(* Logix 5000 project; controller Sucrose_Main Emulate 5570 rev 20.12; software revision 20.01; part 25 of 30 *)
(* tags used below, declared in another part *)
   Alarm_ACK_Master_Timer : TIMER;
   CIPRemote : Area_Program;
   CR13582_AOI : QSI_Discrete_Device;   // CR-13582 SUCROSE RECEIVING PUMP #1 SEAL WATER VALVE
   CR13584_AOI : QSI_Discrete_Device;   // CR-13584 SUCROSE RECEIVING PUMP #2 SEAL WATER VALVE
   DI_E25_2 : ALIAS FOR FLX_E25:2:I;   // Discrete Input EN2T_FLX 192.168.1.25
   DI_E25_3 : ALIAS FOR FLX_E25:3:I;   // Discrete Input EN2T_FLX 192.168.1.25
   DO_E25_4 : ALIAS FOR FLX_E25:4:O;   // Discrete Output EN2T_FLX 192.168.1.25
   DO_E25_5 : ALIAS FOR FLX_E25:5:O;   // Discrete Output EN2T_FLX 192.168.1.25
   FV230001_AOI : QSI_Flow_Valve;   // FV-23-00-01 LAUNCH PIG VALVE V1
   FV230002_AOI : QSI_Flow_Valve;   // FV-23-00-02 LAUNCH PIG VALVE V2
   FV2300031_AOI : QSI_Flow_Valve;   // FV-23-00-03_1 MOVE PIG BACKWARDS INTO CIP/PRODUCTION POSITION
   FV2300032_AOI : QSI_Flow_Valve;   // FV-23-00-03_2 MOVE PIG FORWARD INTO LAUNCHING POSITION
   FV230004_AOI : QSI_Flow_Valve;   // FV-23-00-04 PIG RETENTION CYLINDER V4.1
   FV230005_AOI : QSI_Flow_Valve;   // FV-23-00-05 PIG RETENTION CYLINDER V4.2
   FV230010_AOI : QSI_Flow_Valve;   // FV-23-00-10-O RECEIVING PUMP #1 TO SUCROSE VALVE MANIFOLD MIX PROOF VALVE OPEN
   FV230020_AOI : QSI_Flow_Valve;   // FV-23-00-20-O RECEIVING PUMP #2 TO SUCROSE VALVE MANIFOLD MIX PROOF VALVE OPEN
   IO_Check : BOOL;
   P230010_AOI : PF525_VFD_E_ENET;   // P-23-00-10 RECEIVING PUMP 1
   P230020_AOI : PF525_VFD_E_ENET;   // P-23-00-20 RECEIVING PUMP 2
   PBL1604002_AOI : QSI_Discrete_Device;   // PBL-16040-02 E-STOP CIRCUIT RESET LIGHT
   PSV230010_AOI : QSI_Flow_Valve;
   PSV230020_AOI : QSI_Flow_Valve;
   Sucrose_MM_Enable : BOOL;
   SucroseCIP_RECEIVING2_REMOTE : CIP_REMOTE;
   SucroseCIP_RECEIVING_LINE_REMOTE : CIP_REMOTE;
   SucroseCIP_RECEIVING_REMOTE : CIP_REMOTE;
   SucroseReceiving : Area_Program;
   TMR_SLOW_PLS1 : TIMER;
   TMR_SLOW_PLS2 : TIMER;

PROGRAM ReceivingArea_EN2T_IO_Discrete_DO_E25_4   (* main routine MainRoutine *)

ROUTINE _00_FV230001   (* ladder *)
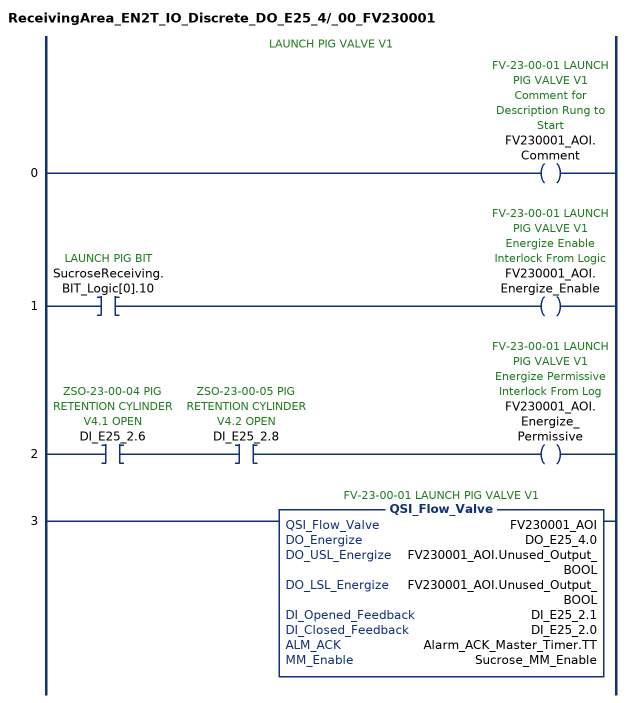
   // LAUNCH PIG VALVE V1
   0: OTE(FV230001_AOI.Comment);
   1: XIC(SucroseReceiving.BIT_Logic[0].10)OTE(FV230001_AOI.Energize_Enable);
   2: XIC(DI_E25_2.6)XIC(DI_E25_2.8)OTE(FV230001_AOI.Energize_Permissive);
   3: QSI_Flow_Valve(FV230001_AOI,DO_E25_4.0,FV230001_AOI.Unused_Output_BOOL,FV230001_AOI.Unused_Output_BOOL,DI_E25_2.1,DI_E25_2.0,Alarm_ACK_Master_Timer.TT,Sucrose_MM_Enable);
END_ROUTINE

ROUTINE _01_FV230002   (* ladder *)
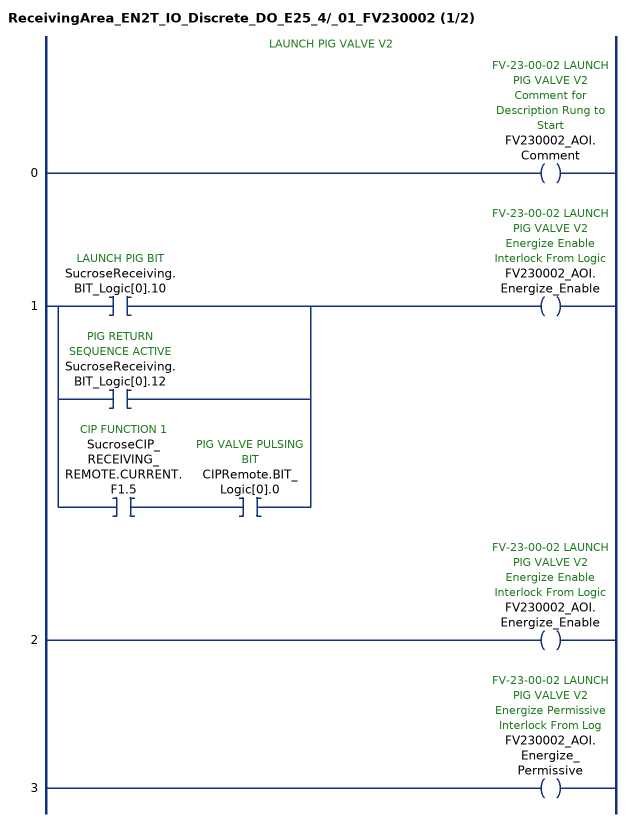
   // LAUNCH PIG VALVE V2
   0: OTE(FV230002_AOI.Comment);
   1: [XIC(SucroseReceiving.BIT_Logic[0].10) ,XIC(SucroseReceiving.BIT_Logic[0].12) ,XIC(SucroseCIP_RECEIVING_REMOTE.CURRENT.F1.5) XIC(CIPRemote.BIT_Logic[0].0) ]OTE(FV230002_AOI.Energize_Enable);
   2: OTE(FV230002_AOI.Energize_Enable);
   3: OTE(FV230002_AOI.Energize_Permissive);
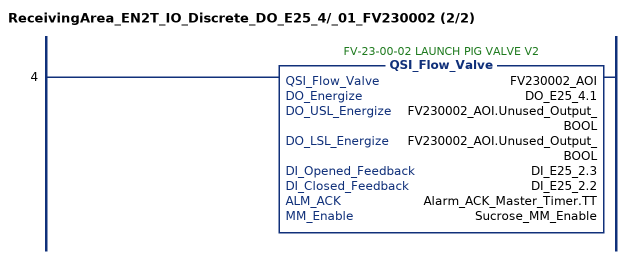
   4: QSI_Flow_Valve(FV230002_AOI,DO_E25_4.1,FV230002_AOI.Unused_Output_BOOL,FV230002_AOI.Unused_Output_BOOL,DI_E25_2.3,DI_E25_2.2,Alarm_ACK_Master_Timer.TT,Sucrose_MM_Enable);
END_ROUTINE

ROUTINE _02_FV230004   (* ladder *)
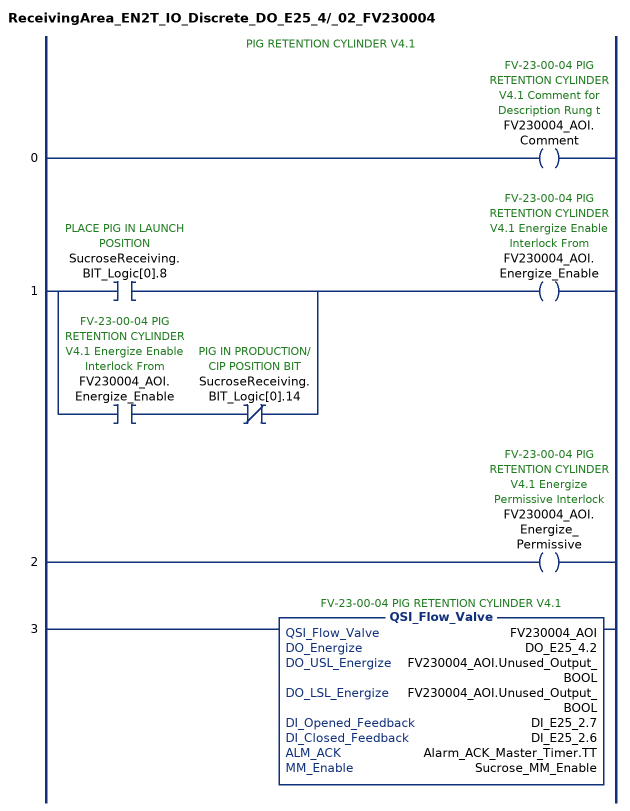
   // PIG RETENTION CYLINDER V4.1
   0: OTE(FV230004_AOI.Comment);
   1: [XIC(SucroseReceiving.BIT_Logic[0].8) ,XIC(FV230004_AOI.Energize_Enable) XIO(SucroseReceiving.BIT_Logic[0].14) ]OTE(FV230004_AOI.Energize_Enable);
   2: OTE(FV230004_AOI.Energize_Permissive);
   3: QSI_Flow_Valve(FV230004_AOI,DO_E25_4.2,FV230004_AOI.Unused_Output_BOOL,FV230004_AOI.Unused_Output_BOOL,DI_E25_2.7,DI_E25_2.6,Alarm_ACK_Master_Timer.TT,Sucrose_MM_Enable);
END_ROUTINE

ROUTINE _03_FV2300031   (* ladder *)
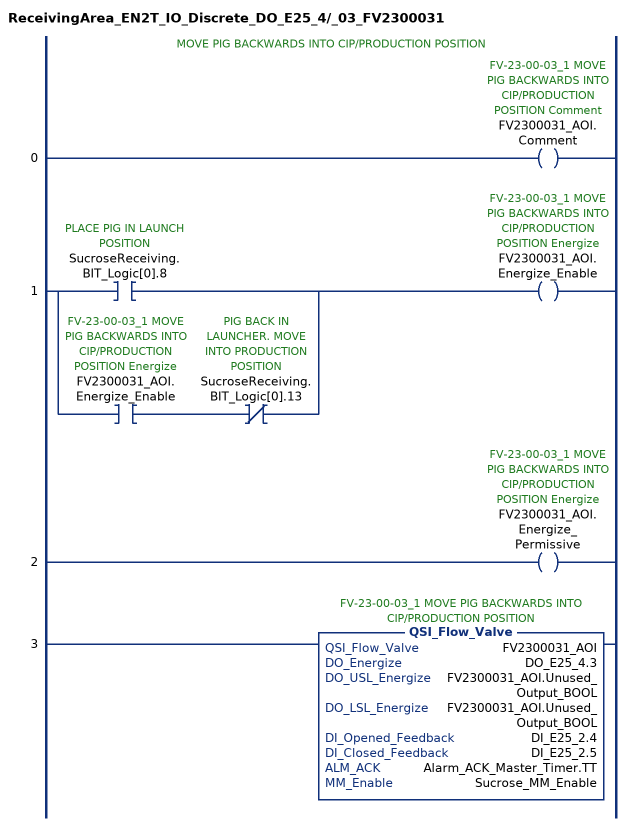
   // MOVE PIG BACKWARDS INTO CIP/PRODUCTION POSITION
   0: OTE(FV2300031_AOI.Comment);
   1: [XIC(SucroseReceiving.BIT_Logic[0].8) ,XIC(FV2300031_AOI.Energize_Enable) XIO(SucroseReceiving.BIT_Logic[0].13) ]OTE(FV2300031_AOI.Energize_Enable);
   2: OTE(FV2300031_AOI.Energize_Permissive);
   3: QSI_Flow_Valve(FV2300031_AOI,DO_E25_4.3,FV2300031_AOI.Unused_Output_BOOL,FV2300031_AOI.Unused_Output_BOOL,DI_E25_2.4,DI_E25_2.5,Alarm_ACK_Master_Timer.TT,Sucrose_MM_Enable);
END_ROUTINE

ROUTINE _04_FV230005   (* ladder *)
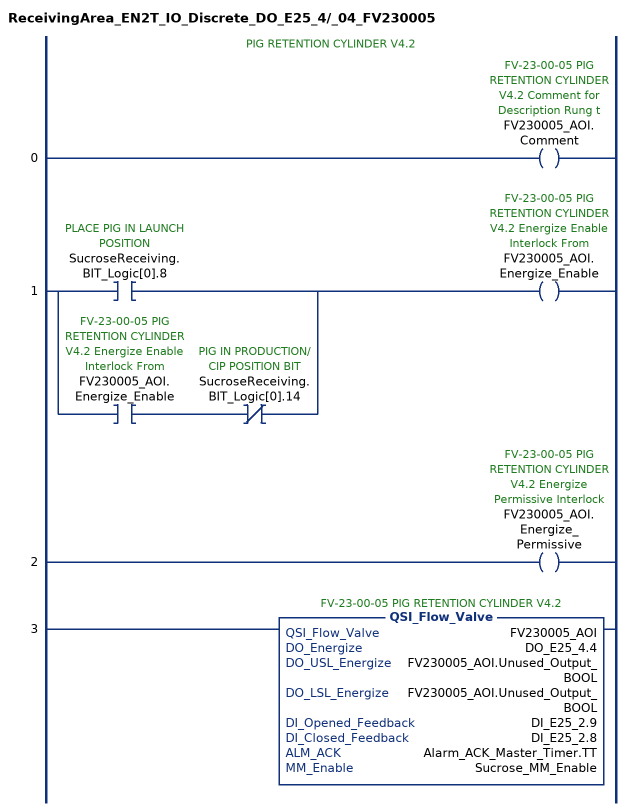
   // PIG RETENTION CYLINDER V4.2
   0: OTE(FV230005_AOI.Comment);
   1: [XIC(SucroseReceiving.BIT_Logic[0].8) ,XIC(FV230005_AOI.Energize_Enable) XIO(SucroseReceiving.BIT_Logic[0].14) ]OTE(FV230005_AOI.Energize_Enable);
   2: OTE(FV230005_AOI.Energize_Permissive);
   3: QSI_Flow_Valve(FV230005_AOI,DO_E25_4.4,FV230005_AOI.Unused_Output_BOOL,FV230005_AOI.Unused_Output_BOOL,DI_E25_2.9,DI_E25_2.8,Alarm_ACK_Master_Timer.TT,Sucrose_MM_Enable);
END_ROUTINE

ROUTINE _05_FV2300032   (* ladder *)
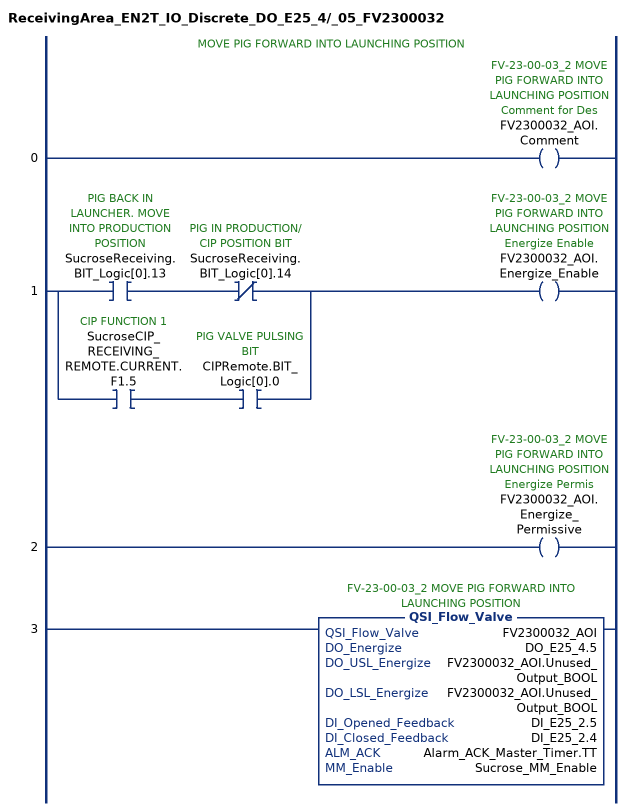
   // MOVE PIG FORWARD INTO LAUNCHING POSITION
   0: OTE(FV2300032_AOI.Comment);
   1: [XIC(SucroseReceiving.BIT_Logic[0].13) XIO(SucroseReceiving.BIT_Logic[0].14) ,XIC(SucroseCIP_RECEIVING_REMOTE.CURRENT.F1.5) XIC(CIPRemote.BIT_Logic[0].0) ]OTE(FV2300032_AOI.Energize_Enable);
   2: OTE(FV2300032_AOI.Energize_Permissive);
   3: QSI_Flow_Valve(FV2300032_AOI,DO_E25_4.5,FV2300032_AOI.Unused_Output_BOOL,FV2300032_AOI.Unused_Output_BOOL,DI_E25_2.5,DI_E25_2.4,Alarm_ACK_Master_Timer.TT,Sucrose_MM_Enable);
END_ROUTINE

ROUTINE _10_PSV230010   (* ladder *)
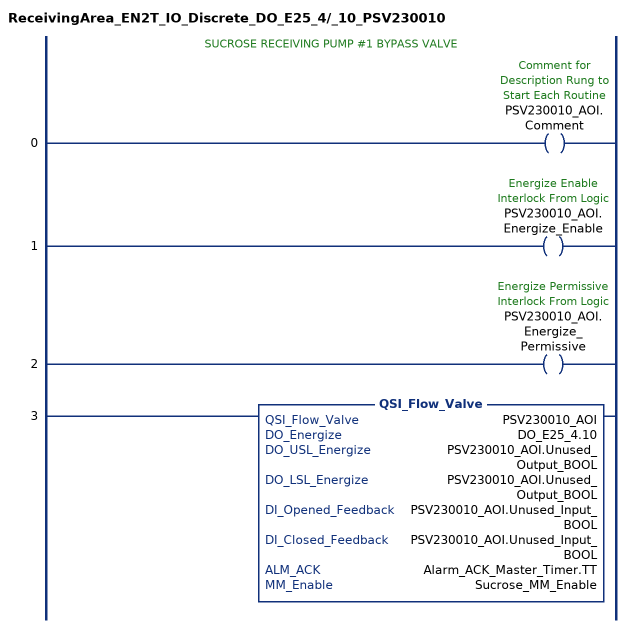
   // SUCROSE RECEIVING PUMP #1 BYPASS VALVE
   0: OTE(PSV230010_AOI.Comment);
   1: OTE(PSV230010_AOI.Energize_Enable);
   2: OTE(PSV230010_AOI.Energize_Permissive);
   3: QSI_Flow_Valve(PSV230010_AOI,DO_E25_4.10,PSV230010_AOI.Unused_Output_BOOL,PSV230010_AOI.Unused_Output_BOOL,PSV230010_AOI.Unused_Input_BOOL,PSV230010_AOI.Unused_Input_BOOL,Alarm_ACK_Master_Timer.TT,Sucrose_MM_Enable);
END_ROUTINE

ROUTINE _11_PSV230020   (* ladder *)
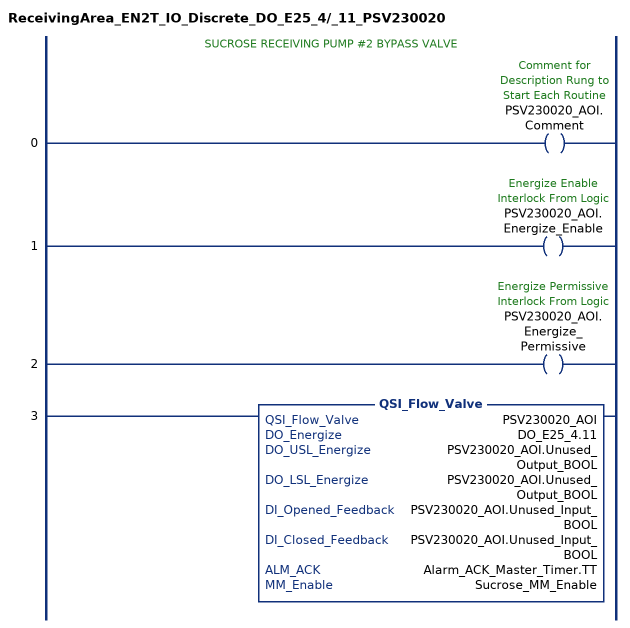
   // SUCROSE RECEIVING PUMP #2 BYPASS VALVE
   0: OTE(PSV230020_AOI.Comment);
   1: OTE(PSV230020_AOI.Energize_Enable);
   2: OTE(PSV230020_AOI.Energize_Permissive);
   3: QSI_Flow_Valve(PSV230020_AOI,DO_E25_4.11,PSV230020_AOI.Unused_Output_BOOL,PSV230020_AOI.Unused_Output_BOOL,PSV230020_AOI.Unused_Input_BOOL,PSV230020_AOI.Unused_Input_BOOL,Alarm_ACK_Master_Timer.TT,Sucrose_MM_Enable);
END_ROUTINE

ROUTINE MainRoutine   (* ladder *)
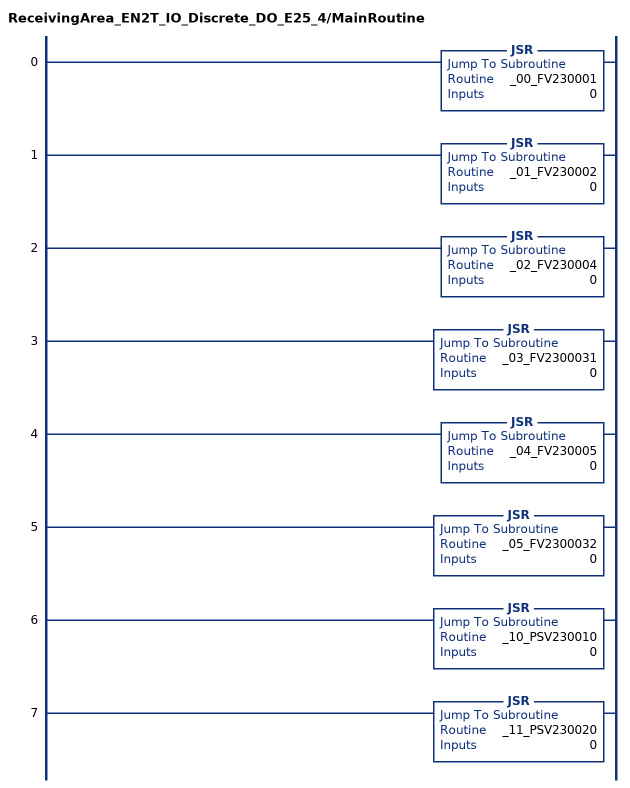
   0: JSR(_00_FV230001,0);
   1: JSR(_01_FV230002,0);
   2: JSR(_02_FV230004,0);
   3: JSR(_03_FV2300031,0);
   4: JSR(_04_FV230005,0);
   5: JSR(_05_FV2300032,0);
   6: JSR(_10_PSV230010,0);
   7: JSR(_11_PSV230020,0);
END_ROUTINE
END_PROGRAM

PROGRAM ReceivingArea_EN2T_IO_Discrete_DO_E25_5   (* main routine MainRoutine *)

ROUTINE _00_FV230010   (* ladder *)
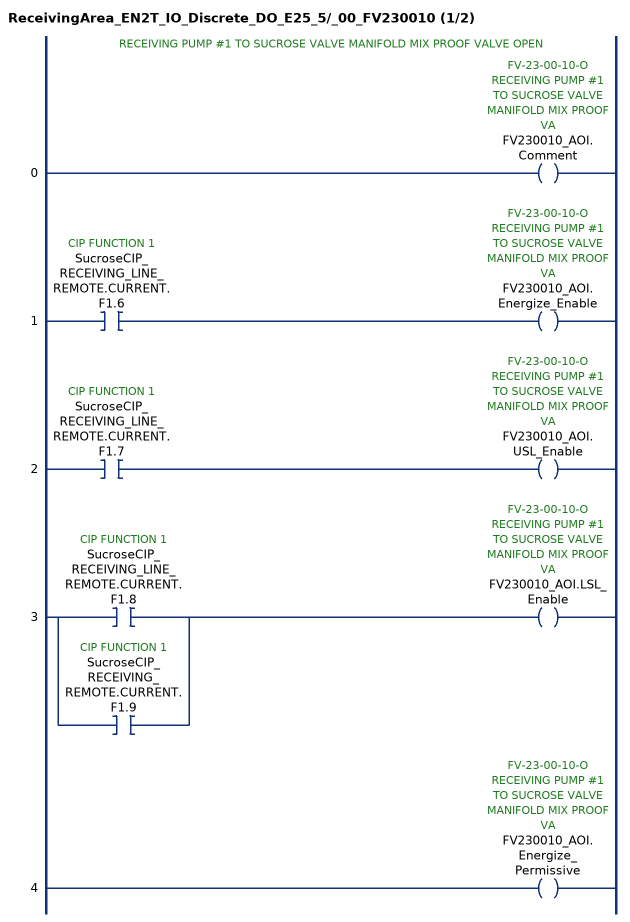
   // RECEIVING PUMP #1 TO SUCROSE VALVE MANIFOLD MIX PROOF VALVE OPEN
   0: OTE(FV230010_AOI.Comment);
   1: XIC(SucroseCIP_RECEIVING_LINE_REMOTE.CURRENT.F1.6)OTE(FV230010_AOI.Energize_Enable);
   2: XIC(SucroseCIP_RECEIVING_LINE_REMOTE.CURRENT.F1.7)OTE(FV230010_AOI.USL_Enable);
   3: [XIC(SucroseCIP_RECEIVING_LINE_REMOTE.CURRENT.F1.8) ,XIC(SucroseCIP_RECEIVING_REMOTE.CURRENT.F1.9) ]OTE(FV230010_AOI.LSL_Enable);
   4: OTE(FV230010_AOI.Energize_Permissive);
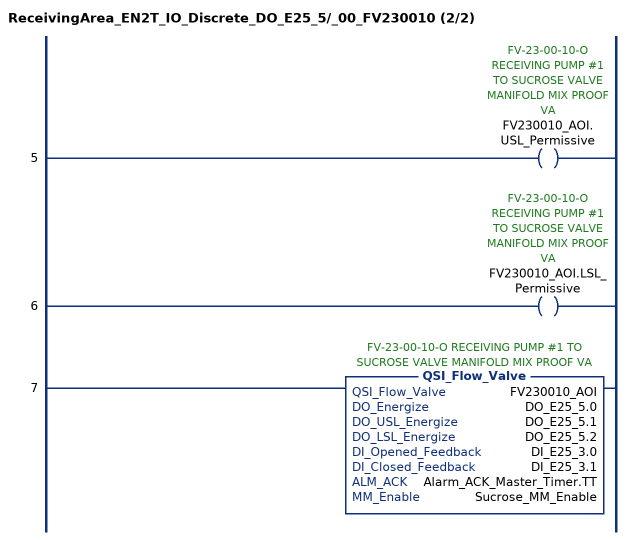
   5: OTE(FV230010_AOI.USL_Permissive);
   6: OTE(FV230010_AOI.LSL_Permissive);
   7: QSI_Flow_Valve(FV230010_AOI,DO_E25_5.0,DO_E25_5.1,DO_E25_5.2,DI_E25_3.0,DI_E25_3.1,Alarm_ACK_Master_Timer.TT,Sucrose_MM_Enable);
END_ROUTINE

ROUTINE _03_FV230020   (* ladder *)
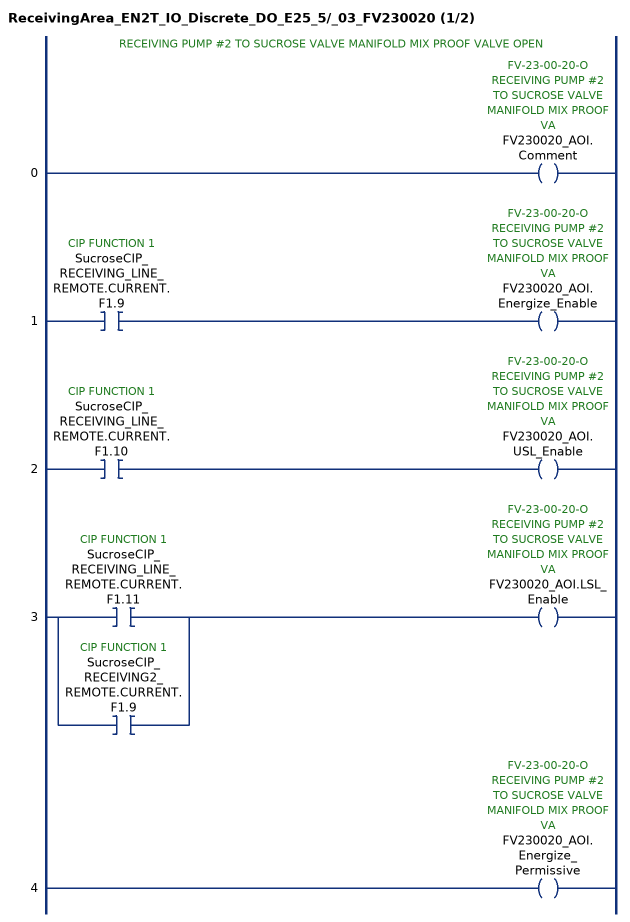
   // RECEIVING PUMP #2 TO SUCROSE VALVE MANIFOLD MIX PROOF VALVE OPEN
   0: OTE(FV230020_AOI.Comment);
   1: XIC(SucroseCIP_RECEIVING_LINE_REMOTE.CURRENT.F1.9)OTE(FV230020_AOI.Energize_Enable);
   2: XIC(SucroseCIP_RECEIVING_LINE_REMOTE.CURRENT.F1.10)OTE(FV230020_AOI.USL_Enable);
   3: [XIC(SucroseCIP_RECEIVING_LINE_REMOTE.CURRENT.F1.11) ,XIC(SucroseCIP_RECEIVING2_REMOTE.CURRENT.F1.9) ]OTE(FV230020_AOI.LSL_Enable);
   4: OTE(FV230020_AOI.Energize_Permissive);
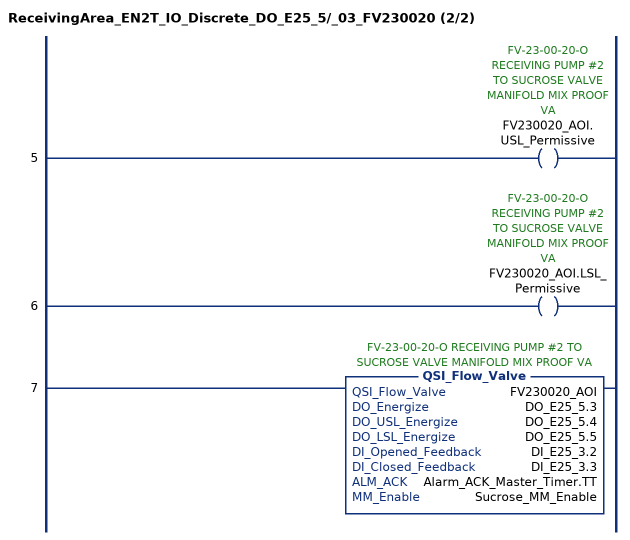
   5: OTE(FV230020_AOI.USL_Permissive);
   6: OTE(FV230020_AOI.LSL_Permissive);
   7: QSI_Flow_Valve(FV230020_AOI,DO_E25_5.3,DO_E25_5.4,DO_E25_5.5,DI_E25_3.2,DI_E25_3.3,Alarm_ACK_Master_Timer.TT,Sucrose_MM_Enable);
END_ROUTINE

ROUTINE _13_PBL1604002   (* ladder *)
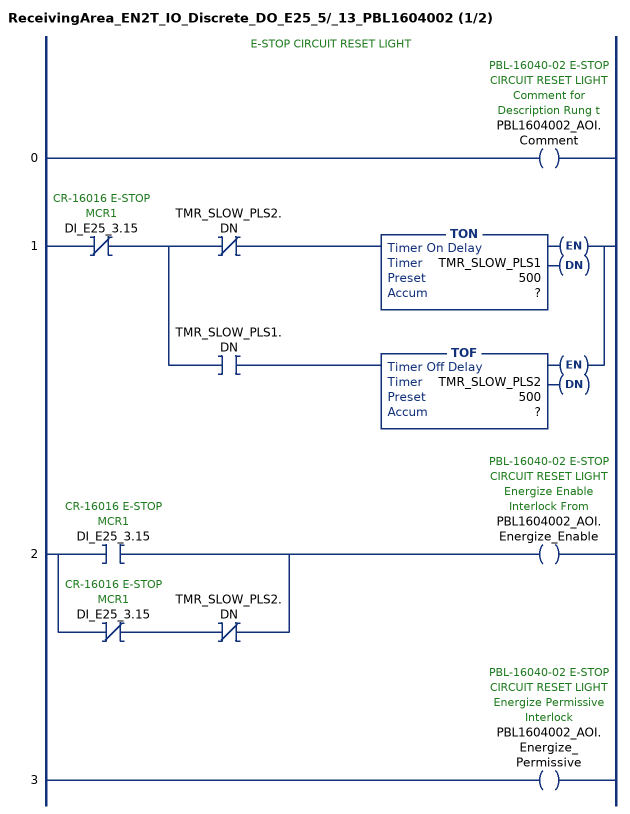
   // E-STOP CIRCUIT RESET LIGHT
   0: OTE(PBL1604002_AOI.Comment);
   1: XIO(DI_E25_3.15)[XIO(TMR_SLOW_PLS2.DN) TON(TMR_SLOW_PLS1,?,?) ,XIC(TMR_SLOW_PLS1.DN) TOF(TMR_SLOW_PLS2,?,?) ];
   2: [XIC(DI_E25_3.15) ,XIO(DI_E25_3.15) XIO(TMR_SLOW_PLS2.DN) ]OTE(PBL1604002_AOI.Energize_Enable);
   3: OTE(PBL1604002_AOI.Energize_Permissive);
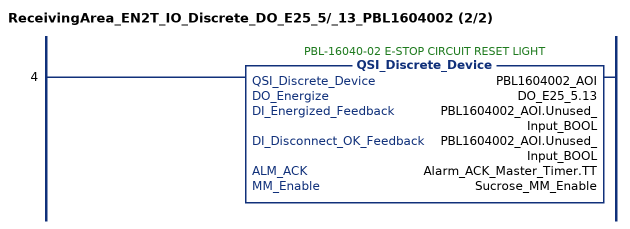
   4: QSI_Discrete_Device(PBL1604002_AOI,DO_E25_5.13,PBL1604002_AOI.Unused_Input_BOOL,PBL1604002_AOI.Unused_Input_BOOL,Alarm_ACK_Master_Timer.TT,Sucrose_MM_Enable);
END_ROUTINE

ROUTINE _14_CR13582   (* ladder *)
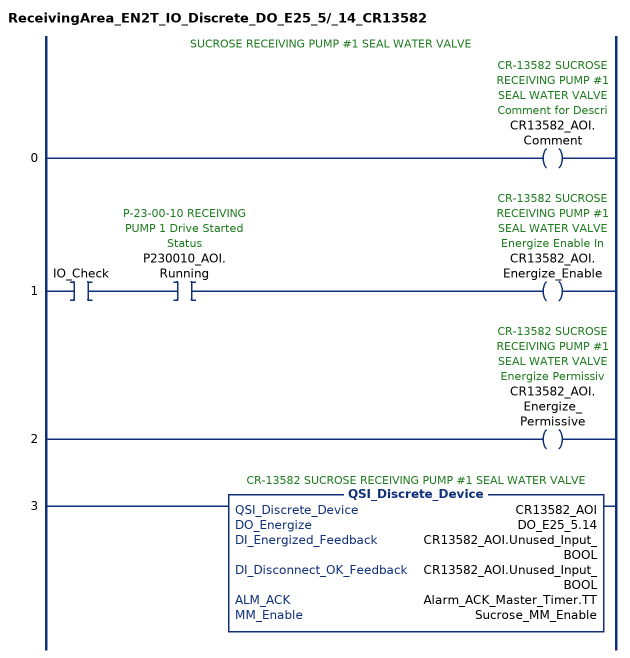
   // SUCROSE RECEIVING PUMP #1 SEAL WATER VALVE
   0: OTE(CR13582_AOI.Comment);
   1: XIC(IO_Check)XIC(P230010_AOI.Running)OTE(CR13582_AOI.Energize_Enable);
   2: OTE(CR13582_AOI.Energize_Permissive);
   3: QSI_Discrete_Device(CR13582_AOI,DO_E25_5.14,CR13582_AOI.Unused_Input_BOOL,CR13582_AOI.Unused_Input_BOOL,Alarm_ACK_Master_Timer.TT,Sucrose_MM_Enable);
END_ROUTINE

ROUTINE _15_CR13584   (* ladder *)
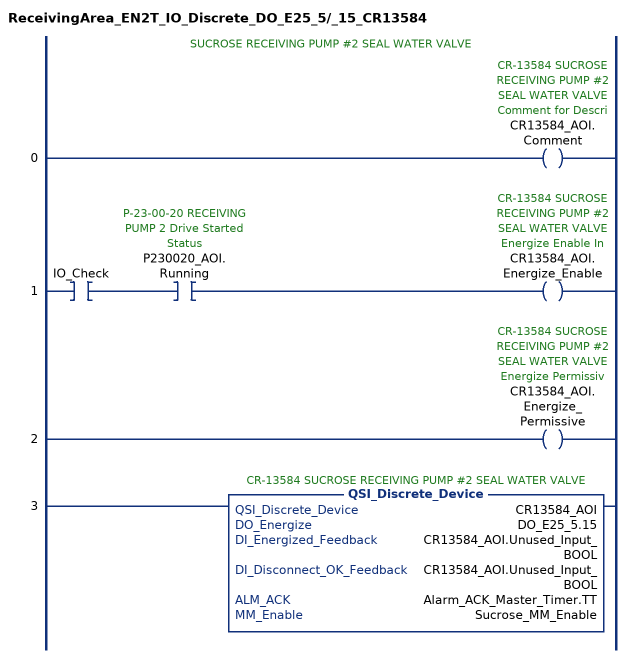
   // SUCROSE RECEIVING PUMP #2 SEAL WATER VALVE
   0: OTE(CR13584_AOI.Comment);
   1: XIC(IO_Check)XIC(P230020_AOI.Running)OTE(CR13584_AOI.Energize_Enable);
   2: OTE(CR13584_AOI.Energize_Permissive);
   3: QSI_Discrete_Device(CR13584_AOI,DO_E25_5.15,CR13584_AOI.Unused_Input_BOOL,CR13584_AOI.Unused_Input_BOOL,Alarm_ACK_Master_Timer.TT,Sucrose_MM_Enable);
END_ROUTINE
